// TIA Portal V20 export
TYPE "typeCmControlNode"
// stored: Namespace Unit1.Em0
   STRUCT
      interlock : "Unit1.Em0.typeCmControlNodeInterlock";
   END_STRUCT;
END_TYPE
